// Mitsubishi GX Works2 project: トッコタッチセンサ動き   PLC: Q03UDV

PROGRAM MAIN
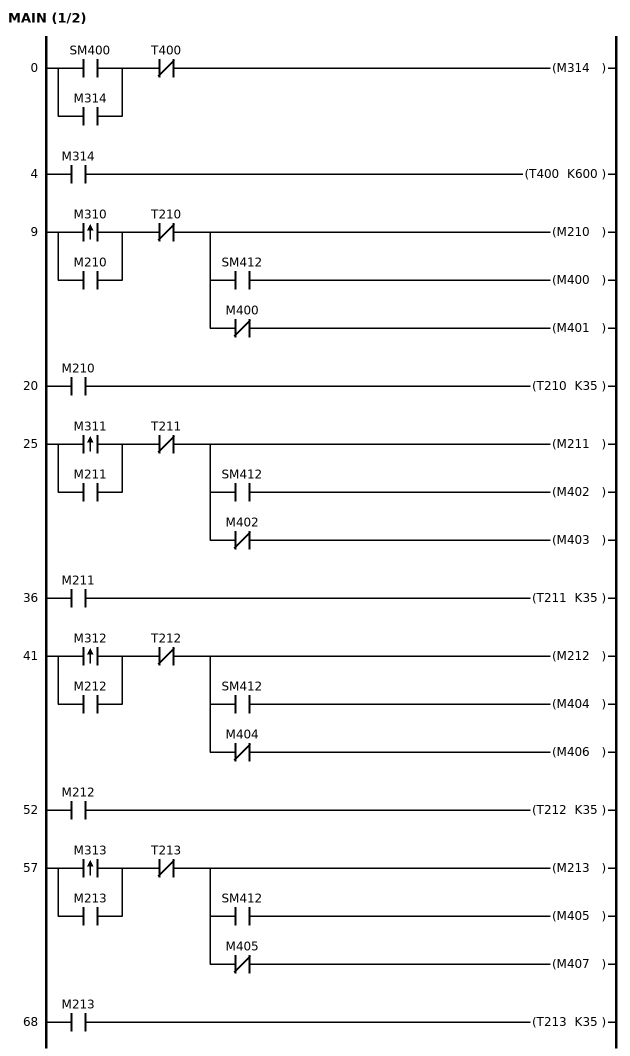
0     LD      SM400
      OR      M314
      ANI     T400
      OUT     M314
4     LD      M314
      OUT     T400 K600
9     LDP     M310
      OR      M210
      ANI     T210
      OUT     M210
      MPS
      AND     SM412
      OUT     M400
      MPP
      ANI     M400
      OUT     M401
20    LD      M210
      OUT     T210 K35
25    LDP     M311
      OR      M211
      ANI     T211
      OUT     M211
      MPS
      AND     SM412
      OUT     M402
      MPP
      ANI     M402
      OUT     M403
36    LD      M211
      OUT     T211 K35
41    LDP     M312
      OR      M212
      ANI     T212
      OUT     M212
      MPS
      AND     SM412
      OUT     M404
      MPP
      ANI     M404
      OUT     M406
52    LD      M212
      OUT     T212 K35
57    LDP     M313
      OR      M213
      ANI     T213
      OUT     M213
      MPS
      AND     SM412
      OUT     M405
      MPP
      ANI     M405
      OUT     M407
68    LD      M213
      OUT     T213 K35
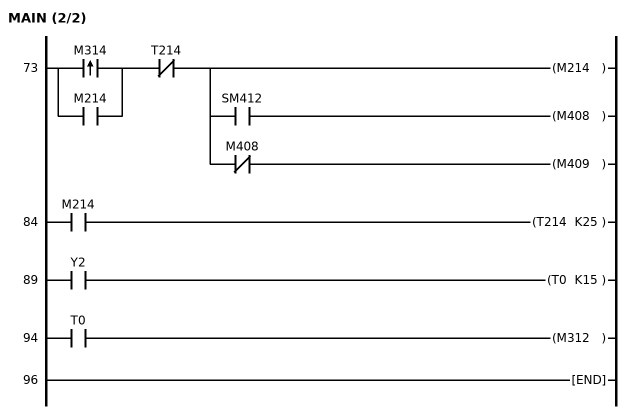
73    LDP     M314
      OR      M214
      ANI     T214
      OUT     M214
      MPS
      AND     SM412
      OUT     M408
      MPP
      ANI     M408
      OUT     M409
84    LD      M214
      OUT     T214 K25
89    LD      Y2
      OUT     T0 K15
94    LD      T0
      OUT     M312
96    END
END_PROGRAM
